FUNCTION_BLOCK FB_lbIOmapping
VAR_INPUT
	iLb	: INT;
	//sNetID	: STRING;
	//nSlaveAddr : UINT;
END_VAR
VAR_OUTPUT
END_VAR
VAR_IN_OUT
	
END_VAR
VAR
	offset	: INT;
END_VAR

offset:= 87+iLb*3;
GVL.lb[iLb].contactor_beltConv					:= G_IO.arDI[offset].Ch[0];
GVL.lb[iLb].valve_stopper[0].extended			:= G_IO.arDI[offset].Ch[1];
GVL.lb[iLb].valve_stopper[0].retracted			:= G_IO.arDI[offset].Ch[2];
GVL.lb[iLb].valve_stopper[1].extended			:= G_IO.arDI[offset].Ch[3];
GVL.lb[iLb].valve_stopper[1].retracted			:= G_IO.arDI[offset].Ch[4];
GVL.lb[iLb].valve_stopper[2].extended			:= G_IO.arDI[offset].Ch[5];
GVL.lb[iLb].valve_stopper[2].retracted			:= G_IO.arDI[offset].Ch[6];
GVL.lb[iLb].valve_stopper[3].extended			:= G_IO.arDI[offset].Ch[7];
GVL.lb[iLb].valve_stopper[3].retracted			:= G_IO.arDI[offset].Ch[8];
GVL.lb[iLb].valve_stopper[4].extended			:= G_IO.arDI[offset].Ch[9];
GVL.lb[iLb].valve_stopper[4].retracted			:= G_IO.arDI[offset].Ch[10];
GVL.lb[iLb].valve_stopper[5].extended			:= G_IO.arDI[offset].Ch[11];
GVL.lb[iLb].valve_stopper[5].retracted			:= G_IO.arDI[offset].Ch[12];
GVL.lb[iLb].photo_sensor[0]						:= G_IO.arDI[offset].Ch[13];
GVL.lb[iLb].photo_sensor[1]						:= G_IO.arDI[offset].Ch[14];
GVL.lb[iLb].photo_sensor[2]						:= G_IO.arDI[offset].Ch[15];



G_IO.arDO[offset].Ch[0]		:= GVL.lb[iLb].power_beltConv;
G_IO.arDO[offset].Ch[1]		:= GVL.lb[iLb].valve_stopper[0].retract;
G_IO.arDO[offset].Ch[2]		:= GVL.lb[iLb].valve_stopper[1].retract;
G_IO.arDO[offset].Ch[3]		:= GVL.lb[iLb].valve_stopper[2].retract;
G_IO.arDO[offset].Ch[4]		:= GVL.lb[iLb].valve_stopper[3].retract;
G_IO.arDO[offset].Ch[5]		:= GVL.lb[iLb].valve_stopper[4].retract;
G_IO.arDO[offset].Ch[6]		:= GVL.lb[iLb].valve_stopper[5].retract;

END_FUNCTION_BLOCK

(* stored: Version 1.1.0.1, ProductVersion 3.1.4024.12
   POU FB_lbIOmapping: Id {4848e81c-3fcd-4cac-8805-1ea8c3359cba}, SpecialFunc None *)
